(* POU GENERAL/xFctCheckNumber, ST *)
FUNCTION xFctCheckNumber : BOOL
VAR_INPUT
	sValue:STRING(255);
	xAlowDoubleSign:BOOL;
END_VAR
VAR
	iCharCount: INT;
	ii: INT;
	sCopyChar: STRING;
	xTmp: BOOL;
	xSyntaxError: BOOL;
	iCountPointChar: INT;
	iCountMinusChar: INT;
	iCountPlusChar: INT;
	iCountExponentChar: INT;
END_VAR
xFctCheckNumber:=FALSE;
iCharCount:=LEN(sValue);
iCountPointChar:=0;
iCountMinusChar:=0;
iCountPlusChar:=0;
iCountExponentChar:=0;
xSyntaxError:=FALSE;
IF (sValue <> '') THEN
	FOR ii:=1 TO iCharCount DO
		sCopyChar:=MID(sValue,1,ii);
		xTmp:=	(sCopyChar = '0') OR (sCopyChar = '1') OR (sCopyChar = '2') OR (sCopyChar = '3') OR (sCopyChar = '4') OR
				(sCopyChar = '5') OR (sCopyChar = '6') OR (sCopyChar = '7') OR (sCopyChar = '8') OR (sCopyChar = '9') OR
				(sCopyChar = '.') OR (sCopyChar = '-') OR (sCopyChar = '+') OR (sCopyChar = 'e') OR (sCopyChar = 'E');
		IF (sCopyChar = '.') THEN
			iCountPointChar:=iCountPointChar + 1;
		END_IF;
		IF (sCopyChar = '-') THEN
			iCountMinusChar:=iCountMinusChar + 1;
		END_IF;
		IF (sCopyChar = '+') THEN
			iCountPlusChar:=iCountPlusChar + 1;
		END_IF;
		IF (sCopyChar = 'e') OR (sCopyChar = 'E') THEN
			iCountExponentChar:=iCountExponentChar + 1;
			IF (iCountMinusChar > 0) THEN
				iCountMinusChar:=iCountMinusChar -1;
			END_IF;
			IF (iCountPlusChar > 0) THEN
				iCountPlusChar:=iCountPlusChar -1;
			END_IF;
		END_IF;
		IF NOT(xTmp) OR (iCountPointChar > 1) OR ((iCountMinusChar > 1) AND NOT(xAlowDoubleSign)) OR ((iCountMinusChar > 2) AND xAlowDoubleSign) OR
		    ((iCountPlusChar > 1) AND NOT(xAlowDoubleSign)) OR ((iCountPlusChar > 2) AND xAlowDoubleSign) OR (iCountExponentChar > 1) THEN
			xSyntaxError:=TRUE;
			EXIT;
		END_IF;
	END_FOR;
ELSE
	xSyntaxError:=TRUE;
END_IF;
xFctCheckNumber:=NOT(xSyntaxError);
END_FUNCTION

(* POU GENERAL/PROFILE/xFctCopyProfileToDataFile, ST *)
FUNCTION xFctCopyProfileToDataFile : BOOL
VAR_INPUT
	sNameOfProfile:STRING(30);
	ptrStProzessData:POINTER TO ST_EXCHG_PARAM_STANDARDPROCESS;
	ptrOnlineChangeData:POINTER TO ST_PROFILEONLINECHANGE_DATA;
	ptrDataFile:POINTER TO ARRAY[1..csiMaxFileLine] OF STRING(csiMaxCharPerLine);
END_VAR
VAR
(* variable *)
	i:INT;
(* Tmp *)
	sTmp:STRING;
END_VAR
(* Init. variable *)
	xFctCopyProfileToDataFile:=FALSE;
	i:=1;

(* copy value *)
	(* Name of the profile *)
		ptrDataFile^[i]:=sNameOfProfile;i:=i+1;
		sTmp:=CONCAT('001:rTorqueLevelHC:=',REAL_TO_STRING(ptrOnlineChangeData^.rTorqueLevelHC));
		ptrDataFile^[i]:=CONCAT(sTmp,';');i:=i+1;
		sTmp:=CONCAT('002:rForceDeflection:=',REAL_TO_STRING(ptrOnlineChangeData^.rForceDeflection));
		ptrDataFile^[i]:=CONCAT(sTmp,';');i:=i+1;
		sTmp:=CONCAT('003:rWorkingSpeedForward:=',REAL_TO_STRING(ptrOnlineChangeData^.rWorkingSpeedForward));
		ptrDataFile^[i]:=CONCAT(sTmp,';');i:=i+1;
		sTmp:=CONCAT('004:rWorkingOffsetBackward:=',REAL_TO_STRING(ptrOnlineChangeData^.rWorkingOffsetBackward));
		ptrDataFile^[i]:=CONCAT(sTmp,';');i:=i+1;
		sTmp:=CONCAT('005:rWorkingSpeedBackward:=',REAL_TO_STRING(ptrOnlineChangeData^.rWorkingSpeedBackward));
		ptrDataFile^[i]:=CONCAT(sTmp,';');i:=i+1;
		sTmp:=CONCAT('006:rWorkingSpindleSpeed:=',REAL_TO_STRING(ptrOnlineChangeData^.rWorkingSpindleSpeed));
		ptrDataFile^[i]:=CONCAT(sTmp,';');i:=i+1;

		sTmp:=CONCAT('007:rPositionLoad:=',REAL_TO_STRING(ptrStProzessData^.rPositionLoad));
		ptrDataFile^[i]:=CONCAT(sTmp,';');i:=i+1;
		sTmp:=CONCAT('008:rPositionStartProc:=',REAL_TO_STRING(ptrStProzessData^.rPositionStartProc));
		ptrDataFile^[i]:=CONCAT(sTmp,';');i:=i+1;
		sTmp:=CONCAT('009:rPositionEndProc:=',REAL_TO_STRING(ptrStProzessData^.rPositionEndProc));
		ptrDataFile^[i]:=CONCAT(sTmp,';');i:=i+1;
		sTmp:=CONCAT('010:rPositionToolChange:=',REAL_TO_STRING(ptrStProzessData^.rPositionToolChange));
		ptrDataFile^[i]:=CONCAT(sTmp,';');i:=i+1;
		sTmp:=CONCAT('011:rInfeedZAxisSpeed:=',REAL_TO_STRING(ptrStProzessData^.rInfeedZAxisSpeed));
		ptrDataFile^[i]:=CONCAT(sTmp,';');i:=i+1;
		sTmp:=CONCAT('012:rInfeedSpindleSpeed:=',REAL_TO_STRING(ptrStProzessData^.rInfeedSpindleSpeed));
		ptrDataFile^[i]:=CONCAT(sTmp,';');i:=i+1;
		sTmp:=CONCAT('013:rOutfeedStrokeAxisSpeed:=',REAL_TO_STRING(ptrStProzessData^.rOutfeedStrokeAxisSpeed));
		ptrDataFile^[i]:=CONCAT(sTmp,';');i:=i+1;
		sTmp:=CONCAT('014:rOutfeedSpindleSpeed:=',REAL_TO_STRING(ptrStProzessData^.rOutfeedSpindleSpeed));
		ptrDataFile^[i]:=CONCAT(sTmp,';');i:=i+1;
		sTmp:=CONCAT('015:rInfeedForceDeflection:=',REAL_TO_STRING(ptrStProzessData^.rInfeedForceDeflection));
		ptrDataFile^[i]:=CONCAT(sTmp,';');i:=i+1;
		sTmp:=CONCAT('016:rInfeedOffsetBackward:=',REAL_TO_STRING(ptrStProzessData^.rInfeedOffsetBackward));
		ptrDataFile^[i]:=CONCAT(sTmp,';');i:=i+1;
		sTmp:=CONCAT('017:iNumberTryInfeed:=',INT_TO_STRING(ptrStProzessData^.iNumberTryInfeed));
		ptrDataFile^[i]:=CONCAT(sTmp,';');i:=i+1;

		sTmp:=CONCAT('018:rProcessMinTime:=',REAL_TO_STRING(ptrStProzessData^.rProcessMinTime));
		ptrDataFile^[i]:=CONCAT(sTmp,';');i:=i+1;
		sTmp:=CONCAT('019:rProcessMaxTime:=',REAL_TO_STRING(ptrStProzessData^.rProcessMaxTime));
		ptrDataFile^[i]:=CONCAT(sTmp,';');i:=i+1;
		sTmp:=CONCAT('020:iHCStartProcPosCounter:=',INT_TO_STRING(ptrStProzessData^.iHCStartProcPosCounter));
		ptrDataFile^[i]:=CONCAT(sTmp,';');i:=i+1;
		sTmp:=CONCAT('021:rDeflectionSensorOffset:=',REAL_TO_STRING(ptrStProzessData^.rDeflectionSensorOffset));
		ptrDataFile^[i]:=CONCAT(sTmp,';');i:=i+1;
		sTmp:=CONCAT('022:rTorqueLevel_Overload:=',REAL_TO_STRING(ptrStProzessData^.rTorqueLevel_Overload));
		ptrDataFile^[i]:=CONCAT(sTmp,';');i:=i+1;

		sTmp:=CONCAT('023:iSparkOutStrokeCount:=',INT_TO_STRING(ptrStProzessData^.iSparkOutStrokeCount));
		ptrDataFile^[i]:=CONCAT(sTmp,';');i:=i+1;
		sTmp:=CONCAT('024:rSparkOutStrokeLength:=',REAL_TO_STRING(ptrStProzessData^.rSparkOutStrokeLength));
		ptrDataFile^[i]:=CONCAT(sTmp,';');i:=i+1;
		sTmp:=CONCAT('025:rSparkOutStrokeSpeed:=',REAL_TO_STRING(ptrStProzessData^.rSparkOutStrokeSpeed));
		ptrDataFile^[i]:=CONCAT(sTmp,';');i:=i+1;
		sTmp:=CONCAT('026:rSparkOutForceDeflection:=',REAL_TO_STRING(ptrStProzessData^.rSparkOutForceDeflection));
		ptrDataFile^[i]:=CONCAT(sTmp,';');i:=i+1;
		sTmp:=CONCAT('027:rSparkOutTorqueLevel:=',REAL_TO_STRING(ptrStProzessData^.rSparkOutTorqueLevel));
		ptrDataFile^[i]:=CONCAT(sTmp,';');i:=i+1;

		sTmp:=CONCAT('028:rPosToolGuid_Up:=',REAL_TO_STRING(ptrStProzessData^.rPosToolGuid_Up));
		ptrDataFile^[i]:=CONCAT(sTmp,';');i:=i+1;
		sTmp:=CONCAT('029:rPosToolGuid_Down:=',REAL_TO_STRING(ptrStProzessData^.rPosToolGuid_Down));
		ptrDataFile^[i]:=CONCAT(sTmp,';');i:=i+1;
		sTmp:=CONCAT('030:rDistanceToolGuide:=',REAL_TO_STRING(ptrStProzessData^.rDistanceToolGuide));
		ptrDataFile^[i]:=CONCAT(sTmp,';');i:=i+1;
		sTmp:=CONCAT('031:rDistanceToolEndPos:=',REAL_TO_STRING(ptrStProzessData^.rDistanceToolEndPos));
		ptrDataFile^[i]:=CONCAT(sTmp,';');i:=i+1;
		sTmp:=CONCAT('032:rLengthTool_Fixed:=',REAL_TO_STRING(ptrStProzessData^.rLengthTool_Fixed));
		ptrDataFile^[i]:=CONCAT(sTmp,';');i:=i+1;
		sTmp:=CONCAT('033:rLengthTool_Work:=',REAL_TO_STRING(ptrStProzessData^.rLengthTool_Work));
		ptrDataFile^[i]:=CONCAT(sTmp,';');i:=i+1;
		sTmp:=CONCAT('034:rLengthToolGuide:=',REAL_TO_STRING(ptrStProzessData^.rLengthToolGuide));
		ptrDataFile^[i]:=CONCAT(sTmp,';');i:=i+1;
		sTmp:=CONCAT('035:rLengthAirTableBoard:=',REAL_TO_STRING(ptrStProzessData^.rLengthAirTableBoard));
		ptrDataFile^[i]:=CONCAT(sTmp,';');i:=i+1;
		sTmp:=CONCAT('036:xConfigActive:=',BOOL_TO_STRING(ptrStProzessData^.xConfigActive));
		ptrDataFile^[i]:=CONCAT(sTmp,';');i:=i+1;

		sTmp:=CONCAT('037:iMaxTorque:=',INT_TO_STRING(ptrStProzessData^.iMaxTorque));
		ptrDataFile^[i]:=CONCAT(sTmp,';');i:=i+1;
		sTmp:=CONCAT('038:rSpeedZAxisForBackward:=',REAL_TO_STRING(ptrStProzessData^.rSpeedZAxisForBackward));
		ptrDataFile^[i]:=CONCAT(sTmp,';');i:=i+1;
		sTmp:=CONCAT('039:rWorkingSpeedOscillation:=',REAL_TO_STRING(ptrStProzessData^.rWorkingSpeedOscillation));
		ptrDataFile^[i]:=CONCAT(sTmp,';');i:=i+1;
		sTmp:=CONCAT('040:rZ1AxisPosSwitchOAxisOff:=',REAL_TO_STRING(ptrStProzessData^.rZ1AxisPosSwitchOAxisOff));
		ptrDataFile^[i]:=CONCAT(sTmp,';');i:=i+1;
		sTmp:=CONCAT('041:xActivateCoolantProcess:=',BOOL_TO_STRING(ptrStProzessData^.xActivateCoolantProcess));
		ptrDataFile^[i]:=CONCAT(sTmp,';');i:=i+1;
		sTmp:=CONCAT('042:rStrokeAxisPosSwitchCoolantOff:=',REAL_TO_STRING(ptrStProzessData^.rStrokeAxisPosSwitchCoolantOff));
		ptrDataFile^[i]:=CONCAT(sTmp,';');i:=i+1;

		sTmp:=CONCAT('043:rCentringPosZ1Axis:=',REAL_TO_STRING(ptrStProzessData^.rCentringPosZ1Axis));
		ptrDataFile^[i]:=CONCAT(sTmp,';');i:=i+1;
		sTmp:=CONCAT('044:rCentringPosSpeedSlowZ1Axis:=',REAL_TO_STRING(ptrStProzessData^.rCentringPosSpeedSlowZ1Axis));
		ptrDataFile^[i]:=CONCAT(sTmp,';');i:=i+1;
		sTmp:=CONCAT('045:rCentringPosSpeedFastZ1Axis:=',REAL_TO_STRING(ptrStProzessData^.rCentringPosSpeedFastZ1Axis));
		ptrDataFile^[i]:=CONCAT(sTmp,';');i:=i+1;
		sTmp:=CONCAT('046:rCentringSpeedSAxis:=',REAL_TO_STRING(ptrStProzessData^.rCentringSpeedSAxis));
		ptrDataFile^[i]:=CONCAT(sTmp,';');i:=i+1;
		sTmp:=CONCAT('047:rCentringSpeedOAxis:=',REAL_TO_STRING(ptrStProzessData^.rCentringSpeedOAxis));
		ptrDataFile^[i]:=CONCAT(sTmp,';');i:=i+1;
		sTmp:=CONCAT('048:rCentringBackStrokeOffsetFirstHC:=',REAL_TO_STRING(ptrStProzessData^.rCentringBackStrokeOffsetFirstHC));
		ptrDataFile^[i]:=CONCAT(sTmp,';');i:=i+1;
		sTmp:=CONCAT('049:rCentringBackStrokeOffsetAfterFirstHC:=',REAL_TO_STRING(ptrStProzessData^.rCentringBackStrokeOffsetAfterFirstHC));
		ptrDataFile^[i]:=CONCAT(sTmp,';');i:=i+1;
		sTmp:=CONCAT('050:rCentringOffsetBeforeLastHC:=',REAL_TO_STRING(ptrStProzessData^.rCentringOffsetBeforeLastHC));
		ptrDataFile^[i]:=CONCAT(sTmp,';');i:=i+1;
		sTmp:=CONCAT('051:rCentringBackStrokeSpeed:=',REAL_TO_STRING(ptrStProzessData^.rCentringBackStrokeSpeed));
		ptrDataFile^[i]:=CONCAT(sTmp,';');i:=i+1;
		sTmp:=CONCAT('052:rCentringTimeHCActive:=',REAL_TO_STRING(ptrStProzessData^.rCentringTimeHCActive));
		ptrDataFile^[i]:=CONCAT(sTmp,';');i:=i+1;
		sTmp:=CONCAT('053:rCentringTimeHCInactive:=',REAL_TO_STRING(ptrStProzessData^.rCentringTimeHCInactive));
		ptrDataFile^[i]:=CONCAT(sTmp,';');i:=i+1;
		sTmp:=CONCAT('054:iCentringNumberMaxHCinWindow:=',INT_TO_STRING(ptrStProzessData^.iCentringNumberMaxHCinWindow));
		ptrDataFile^[i]:=CONCAT(sTmp,';');i:=i+1;
		sTmp:=CONCAT('055:rCentringHCWindow:=',REAL_TO_STRING(ptrStProzessData^.rCentringHCWindow));
		ptrDataFile^[i]:=CONCAT(sTmp,';');i:=i+1;
		sTmp:=CONCAT('056:rCentringForceDeflection:=',REAL_TO_STRING(ptrStProzessData^.rCentringForceDeflection));
		ptrDataFile^[i]:=CONCAT(sTmp,';');i:=i+1;
		sTmp:=CONCAT('057:rCentringOffsetBackward:=',REAL_TO_STRING(ptrStProzessData^.rCentringOffsetBackward));
		ptrDataFile^[i]:=CONCAT(sTmp,';');i:=i+1;
		sTmp:=CONCAT('058:rCenteringDeflectionSensorOffset:=',REAL_TO_STRING(ptrStProzessData^.rCenteringDeflectionSensorOffset));
		ptrDataFile^[i]:=CONCAT(sTmp,';');i:=i+1;
		sTmp:=CONCAT('059:rCentringOffsetSlowToFastZSpeed:=',REAL_TO_STRING(ptrStProzessData^.rCentringOffsetSlowToFastZSpeed));
		ptrDataFile^[i]:=CONCAT(sTmp,';');i:=i+1;
		sTmp:=CONCAT('060:iCentringSelectProcess:=',INT_TO_STRING(ptrStProzessData^.iCentringSelectProcess));
		ptrDataFile^[i]:=CONCAT(sTmp,';');i:=i+1;
		sTmp:=CONCAT('061:xPositionEndProcIncOnOff:=',BOOL_TO_STRING(ptrStProzessData^.xPositionEndProcIncOnOff));
		ptrDataFile^[i]:=CONCAT(sTmp,';');i:=i+1;
		sTmp:=CONCAT('062:rPositionEndProcMaxInc:=',REAL_TO_STRING(ptrStProzessData^.rPositionEndProcMaxInc));
		ptrDataFile^[i]:=CONCAT(sTmp,';');i:=i+1;
		sTmp:=CONCAT('063:rPositionEndProInc:=',REAL_TO_STRING(ptrStProzessData^.rPositionEndProInc));
		ptrDataFile^[i]:=CONCAT(sTmp,';');i:=i+1;

		sTmp:=CONCAT('064:iWorkControlType:=',INT_TO_STRING(ptrStProzessData^.iWorkControlType));
		ptrDataFile^[i]:=CONCAT(sTmp,';');i:=i+1;
		sTmp:=CONCAT('065:rZ_PID_Torque:=',REAL_TO_STRING(ptrStProzessData^.rZ_PID_Torque));
		ptrDataFile^[i]:=CONCAT(sTmp,';');i:=i+1;
		sTmp:=CONCAT('066:rZ_PID_MinSpeed:=',REAL_TO_STRING(ptrStProzessData^.rZ_PID_MinSpeed));
		ptrDataFile^[i]:=CONCAT(sTmp,';');i:=i+1;
		sTmp:=CONCAT('067:rZ_PID_MaxSpeed:=',REAL_TO_STRING(ptrStProzessData^.rZ_PID_MaxSpeed));
		ptrDataFile^[i]:=CONCAT(sTmp,';');i:=i+1;
		sTmp:=CONCAT('068:rZ_PID_Kp:=',REAL_TO_STRING(ptrStProzessData^.rZ_PID_Kp));
		ptrDataFile^[i]:=CONCAT(sTmp,';');i:=i+1;
		sTmp:=CONCAT('069:rZ_PID_Ki:=',REAL_TO_STRING(ptrStProzessData^.rZ_PID_Ki));
		ptrDataFile^[i]:=CONCAT(sTmp,';');i:=i+1;
		sTmp:=CONCAT('070:rZ_PID_Kd:=',REAL_TO_STRING(ptrStProzessData^.rZ_PID_Kd));
		ptrDataFile^[i]:=CONCAT(sTmp,';');i:=i+1;
		sTmp:=CONCAT('071:iZ_PID_FilterM:=',INT_TO_STRING(ptrStProzessData^.iZ_PID_FilterM));
		ptrDataFile^[i]:=CONCAT(sTmp,';');i:=i+1;
		sTmp:=CONCAT('072:rZ_D_Kd:=',REAL_TO_STRING(ptrStProzessData^.rZ_D_Kd));
		ptrDataFile^[i]:=CONCAT(sTmp,';');i:=i+1;
		sTmp:=CONCAT('073:iZ_D_FilterM:=',INT_TO_STRING(ptrStProzessData^.iZ_D_FilterM));
		ptrDataFile^[i]:=CONCAT(sTmp,';');i:=i+1;

		sTmp:=CONCAT('074:rSuspensionBubblerSpeed:=',REAL_TO_STRING(ptrStProzessData^.rSuspensionBubblerSpeed));
		ptrDataFile^[i]:=CONCAT(sTmp,';');i:=i+1;
		sTmp:=CONCAT('075:rSuspensionFeederSpeed:=',REAL_TO_STRING(ptrStProzessData^.rSuspensionFeederSpeed));
		ptrDataFile^[i]:=CONCAT(sTmp,';');i:=i+1;

		sTmp:=CONCAT('076:rOutfeedStrokeAxisSpeedSlow:=',REAL_TO_STRING(ptrStProzessData^.rOutfeedStrokeAxisSpeedSlow));
		ptrDataFile^[i]:=CONCAT(sTmp,';');i:=i+1;
		sTmp:=CONCAT('077:rZ1AxisPosSwitchFastVel:=',REAL_TO_STRING(ptrStProzessData^.rZ1AxisPosSwitchFastVel));
		ptrDataFile^[i]:=CONCAT(sTmp,';');i:=i+1;
		sTmp:=CONCAT('078:rZ1AxisOffsetStartRecordTorque:=',REAL_TO_STRING(ptrStProzessData^.rZ1AxisOffsetStartRecordTorque));
		ptrDataFile^[i]:=CONCAT(sTmp,';');i:=i+1;

		sTmp:=CONCAT('079:xCentringEndProcIncOnOff:=',BOOL_TO_STRING(ptrStProzessData^.xCentringEndProcIncOnOff));
		ptrDataFile^[i]:=CONCAT(sTmp,';');i:=i+1;
		sTmp:=CONCAT('080:rCentringEndProInc:=',REAL_TO_STRING(ptrStProzessData^.rCentringEndProInc));
		ptrDataFile^[i]:=CONCAT(sTmp,';');i:=i+1;

		sTmp:=CONCAT('081:rWorkingSpindleSpeedMinMax:=',REAL_TO_STRING(ptrStProzessData^.rWorkingSpindleSpeedMinMax));
		ptrDataFile^[i]:=CONCAT(sTmp,';');i:=i+1;
		sTmp:=CONCAT('082:rO_Ctrl_TorquePercent_OFF:=',REAL_TO_STRING(ptrStProzessData^.rO_Ctrl_TorquePercent_OFF));
		ptrDataFile^[i]:=CONCAT(sTmp,';');i:=i+1;
		sTmp:=CONCAT('083:rO_Ctrl_HystereseOffset:=',REAL_TO_STRING(ptrStProzessData^.rO_Ctrl_HystereseOffset));
		ptrDataFile^[i]:=CONCAT(sTmp,';');i:=i+1;

		sTmp:=CONCAT('084:rZPositionCylindricalArea:=',REAL_TO_STRING(ptrStProzessData^.rZPositionCylindricalArea));
		ptrDataFile^[i]:=CONCAT(sTmp,';');i:=i+1;
		sTmp:=CONCAT('085:rZMinThresholdTroqueEndProcess:=',REAL_TO_STRING(ptrStProzessData^.rZMinThresholdTroqueEndProcess));
		ptrDataFile^[i]:=CONCAT(sTmp,';');i:=i+1;

		sTmp:=CONCAT('086:rDistProgressStroke:=',REAL_TO_STRING(ptrStProzessData^.rDistProgressStroke));
		ptrDataFile^[i]:=CONCAT(sTmp,';');i:=i+1;
		sTmp:=CONCAT('087:iProgressStrokeStartTorque:=',INT_TO_STRING(ptrStProzessData^.iProgressStrokeStartTorque));
		ptrDataFile^[i]:=CONCAT(sTmp,';');i:=i+1;
		sTmp:=CONCAT('088:rProgressStrokeStopOffset:=',REAL_TO_STRING(ptrStProzessData^.rProgressStrokeStopOffset));
		ptrDataFile^[i]:=CONCAT(sTmp,';');i:=i+1;
		sTmp:=CONCAT('089:iCleanNozzleMode:=',INT_TO_STRING(ptrStProzessData^.iCleanNozzleMode));
		ptrDataFile^[i]:=CONCAT(sTmp,';');i:=i+1;
		sTmp:=CONCAT('090:ioutfeedstrokecontroller:=',INT_TO_STRING(ptrStProzessData^.iOutfeedStrokeController));
		ptrDataFile^[i]:=CONCAT(sTmp,';');i:=i+1;
		sTmp:=CONCAT('091:isparkoutcontroller:=',INT_TO_STRING(ptrStProzessData^.iSparkOutController));
		ptrDataFile^[i]:=CONCAT(sTmp,';');i:=i+1;

	(* add empty line to set the end *)
	ptrDataFile^[i]:='';

	(* confirm copy *)
	xFctCopyProfileToDataFile:=TRUE;
END_FUNCTION

(* POU GENERAL/PROFILE/xFctSetDefaultValueStaticProfile, ST *)
FUNCTION xFctSetDefaultValueStaticProfile : BOOL
VAR_INPUT
	ptrT_DefaultProfileParameter:POINTER TO ARRAY [1..1] OF ST_RETAIN_DATA_PROFILEPARAMETER;
END_VAR
VAR
(* variable *)
	ii:INT;
END_VAR
	(* Init. value *)
	xFctSetDefaultValueStaticProfile:=FALSE;
	FOR ii:=1 TO 1 DO
		ptrT_DefaultProfileParameter^[ii].T_ProfileOnlineChange.rTorqueLevelHC:=80.0;
		ptrT_DefaultProfileParameter^[ii].T_ProfileOnlineChange.rForceDeflection:=18.0;
		ptrT_DefaultProfileParameter^[ii].T_ProfileOnlineChange.rWorkingSpeedForward:=100.0;
		ptrT_DefaultProfileParameter^[ii].T_ProfileOnlineChange.rWorkingOffsetBackward:=0.0;
		ptrT_DefaultProfileParameter^[ii].T_ProfileOnlineChange.rWorkingSpeedBackward:=0.5;
		ptrT_DefaultProfileParameter^[ii].T_ProfileOnlineChange.rWorkingSpindleSpeed:=6000.0;

		ptrT_DefaultProfileParameter^[ii].T_ProzessData.rPositionLoad:=-446.0;
		ptrT_DefaultProfileParameter^[ii].T_ProzessData.rPositionStartProc:=-410.0;
		ptrT_DefaultProfileParameter^[ii].T_ProzessData.rPositionEndProc:=-80.0;
		ptrT_DefaultProfileParameter^[ii].T_ProzessData.rPositionToolChange:=-510.0;
		ptrT_DefaultProfileParameter^[ii].T_ProzessData.rInfeedZAxisSpeed:=50.0;
		ptrT_DefaultProfileParameter^[ii].T_ProzessData.rInfeedSpindleSpeed:=500.0;
		ptrT_DefaultProfileParameter^[ii].T_ProzessData.rOutfeedStrokeAxisSpeed:=250.0;
		ptrT_DefaultProfileParameter^[ii].T_ProzessData.rOutfeedSpindleSpeed:=500.0;
		ptrT_DefaultProfileParameter^[ii].T_ProzessData.rInfeedForceDeflection:=5.0;
		ptrT_DefaultProfileParameter^[ii].T_ProzessData.rInfeedOffsetBackward:=-10.0;
		ptrT_DefaultProfileParameter^[ii].T_ProzessData.iNumberTryInfeed:=5;

		ptrT_DefaultProfileParameter^[ii].T_ProzessData.rProcessMinTime:=5.0;
		ptrT_DefaultProfileParameter^[ii].T_ProzessData.rProcessMaxTime:=120.0;
		ptrT_DefaultProfileParameter^[ii].T_ProzessData.iHCStartProcPosCounter:=3;
		ptrT_DefaultProfileParameter^[ii].T_ProzessData.rDeflectionSensorOffset:=0.2;
		ptrT_DefaultProfileParameter^[ii].T_ProzessData.rTorqueLevel_Overload:=60.0;

		ptrT_DefaultProfileParameter^[ii].T_ProzessData.iSparkOutStrokeCount:=2;
		ptrT_DefaultProfileParameter^[ii].T_ProzessData.rSparkOutStrokeLength:=-20.0;
		ptrT_DefaultProfileParameter^[ii].T_ProzessData.rSparkOutStrokeSpeed:=200.0;
		ptrT_DefaultProfileParameter^[ii].T_ProzessData.rSparkOutForceDeflection:=80.0;
		ptrT_DefaultProfileParameter^[ii].T_ProzessData.rSparkOutTorqueLevel:=20.0;

		ptrT_DefaultProfileParameter^[ii].T_ProzessData.rPosToolGuid_Up:=210;
		ptrT_DefaultProfileParameter^[ii].T_ProzessData.rPosToolGuid_Down:=185;
		ptrT_DefaultProfileParameter^[ii].T_ProzessData.rDistanceToolGuide:=4.5;
		ptrT_DefaultProfileParameter^[ii].T_ProzessData.rDistanceToolEndPos:=4.5;
		ptrT_DefaultProfileParameter^[ii].T_ProzessData.rLengthTool_Fixed:=450.0;
		ptrT_DefaultProfileParameter^[ii].T_ProzessData.rLengthTool_Work:=325.0;
		ptrT_DefaultProfileParameter^[ii].T_ProzessData.rLengthToolGuide:=10.0;
		ptrT_DefaultProfileParameter^[ii].T_ProzessData.rLengthAirTableBoard:=33.0;
		ptrT_DefaultProfileParameter^[ii].T_ProzessData.xConfigActive:=FALSE;

		ptrT_DefaultProfileParameter^[ii].T_ProzessData.iMaxTorque:=130;
		ptrT_DefaultProfileParameter^[ii].T_ProzessData.rSpeedZAxisForBackward:=1.0;
		ptrT_DefaultProfileParameter^[ii].T_ProzessData.rWorkingSpeedOscillation:=0.0;
		ptrT_DefaultProfileParameter^[ii].T_ProzessData.rZ1AxisPosSwitchOAxisOff:=0.0;
		ptrT_DefaultProfileParameter^[ii].T_ProzessData.xActivateCoolantProcess:=FALSE;
		ptrT_DefaultProfileParameter^[ii].T_ProzessData.rStrokeAxisPosSwitchCoolantOff:=-300.0;

		ptrT_DefaultProfileParameter^[ii].T_ProzessData.rCentringPosZ1Axis:=-400.0;
		ptrT_DefaultProfileParameter^[ii].T_ProzessData.rCentringPosSpeedSlowZ1Axis:=20.0;
		ptrT_DefaultProfileParameter^[ii].T_ProzessData.rCentringPosSpeedFastZ1Axis:=50.0;
		ptrT_DefaultProfileParameter^[ii].T_ProzessData.rCentringSpeedSAxis:=500.0;
		ptrT_DefaultProfileParameter^[ii].T_ProzessData.rCentringSpeedOAxis:=40.0;
		ptrT_DefaultProfileParameter^[ii].T_ProzessData.rCentringBackStrokeOffsetFirstHC:=-5.0;
		ptrT_DefaultProfileParameter^[ii].T_ProzessData.rCentringBackStrokeOffsetAfterFirstHC:=-15.0;
		ptrT_DefaultProfileParameter^[ii].T_ProzessData.rCentringOffsetBeforeLastHC:=-3.0;
		ptrT_DefaultProfileParameter^[ii].T_ProzessData.rCentringBackStrokeSpeed:=10.0;
		ptrT_DefaultProfileParameter^[ii].T_ProzessData.rCentringTimeHCActive:=5.0;
		ptrT_DefaultProfileParameter^[ii].T_ProzessData.rCentringTimeHCInactive:=0.5;
		ptrT_DefaultProfileParameter^[ii].T_ProzessData.iCentringNumberMaxHCinWindow:=5;
		ptrT_DefaultProfileParameter^[ii].T_ProzessData.rCentringHCWindow:=0.5;
		ptrT_DefaultProfileParameter^[ii].T_ProzessData.rCentringForceDeflection:=20.0;
		ptrT_DefaultProfileParameter^[ii].T_ProzessData.rCentringOffsetBackward:=-1.0;
		ptrT_DefaultProfileParameter^[ii].T_ProzessData.rCenteringDeflectionSensorOffset:=0.3;
		ptrT_DefaultProfileParameter^[ii].T_ProzessData.rCentringOffsetSlowToFastZSpeed:=40.0;
		ptrT_DefaultProfileParameter^[ii].T_ProzessData.iCentringSelectProcess:=1;
		ptrT_DefaultProfileParameter^[ii].T_ProzessData.xPositionEndProcIncOnOff:=0;
		ptrT_DefaultProfileParameter^[ii].T_ProzessData.rPositionEndProcMaxInc:=-10.0;
		ptrT_DefaultProfileParameter^[ii].T_ProzessData.rPositionEndProInc:=0.2;
		ptrT_DefaultProfileParameter^[ii].T_ProzessData.rOutfeedStrokeAxisSpeedSlow:=2.0;
		ptrT_DefaultProfileParameter^[ii].T_ProzessData.rZ1AxisPosSwitchFastVel:=0.0;
		ptrT_DefaultProfileParameter^[ii].T_ProzessData.rZ1AxisOffsetStartRecordTorque:=0.0;
		ptrT_DefaultProfileParameter^[ii].T_ProzessData.xCentringEndProcIncOnOff:=0;
		ptrT_DefaultProfileParameter^[ii].T_ProzessData.rCentringEndProInc:=0.2;
		ptrT_DefaultProfileParameter^[ii].T_ProzessData.rWorkingSpindleSpeedMinMax:=6000.0;
		ptrT_DefaultProfileParameter^[ii].T_ProzessData.rO_Ctrl_TorquePercent_OFF:=100.0;
		ptrT_DefaultProfileParameter^[ii].T_ProzessData.rO_Ctrl_HystereseOffset:=10.0;
		ptrT_DefaultProfileParameter^[ii].T_ProzessData.rZPositionCylindricalArea:=-240.0;
		ptrT_DefaultProfileParameter^[ii].T_ProzessData.rZMinThresholdTroqueEndProcess:=12.0;

		ptrT_DefaultProfileParameter^[ii].T_ProzessData.iWorkControlType:=1;
		ptrT_DefaultProfileParameter^[ii].T_ProzessData.rZ_PID_Torque:=50.0;
		ptrT_DefaultProfileParameter^[ii].T_ProzessData.rZ_PID_MinSpeed:=2.0;
		ptrT_DefaultProfileParameter^[ii].T_ProzessData.rZ_PID_MaxSpeed:=40.0;
		ptrT_DefaultProfileParameter^[ii].T_ProzessData.rZ_PID_Kp:=2.0;
		ptrT_DefaultProfileParameter^[ii].T_ProzessData.rZ_PID_Ki:=0.5;
		ptrT_DefaultProfileParameter^[ii].T_ProzessData.rZ_PID_Kd:=0.01;
		ptrT_DefaultProfileParameter^[ii].T_ProzessData.iZ_PID_FilterM:=20;
		ptrT_DefaultProfileParameter^[ii].T_ProzessData.rZ_D_Kd:=0.01;
		ptrT_DefaultProfileParameter^[ii].T_ProzessData.iZ_D_FilterM:=20;

		ptrT_DefaultProfileParameter^[ii].T_ProzessData.rSuspensionBubblerSpeed:=20.0;
		ptrT_DefaultProfileParameter^[ii].T_ProzessData.rSuspensionFeederSpeed:=20.0;

		ptrT_DefaultProfileParameter^[ii].T_ProzessData.rDistProgressStroke:=0.0;
		ptrT_DefaultProfileParameter^[ii].T_ProzessData.iProgressStrokeStartTorque:=0;
		ptrT_DefaultProfileParameter^[ii].T_ProzessData.rProgressStrokeStopOffset:=0.0;
		ptrT_DefaultProfileParameter^[ii].T_ProzessData.iCleanNozzleMode:=0;
		ptrT_DefaultProfileParameter^[ii].T_ProzessData.iOutfeedStrokeController:=0;
		ptrT_DefaultProfileParameter^[ii].T_ProzessData.iSparkOutController:=0;

	END_FOR;
	(* Confirm Default setting *)
	xFctSetDefaultValueStaticProfile:=TRUE;
END_FUNCTION

(* POU GENERAL/FB_PASSWORD, ST *)
FUNCTION_BLOCK FB_PASSWORD
VAR_INPUT
END_VAR
VAR_IN_OUT
	T_Password:ST_PASSWORD;
	T_HDD:ST_HDD;
END_VAR
VAR_OUTPUT
END_VAR
VAR
	RisingEdgeReset: R_TRIG;
	xConfirmResetFB: BOOL;
	TimerFileLocked: TON;
	RisingEdgeExecute: R_TRIG;
	TimerOut: TON;
	xTmp: BOOL;
	tTimeOut: TIME;
	iStepFunction: INT;
	xReadPassword: BOOL;
	sDeleteData: ARRAY[1..csiMaxFileLine] OF STRING(csiMaxCharPerLine);
	sTmp:STRING(255);
	xWritePassword: BOOL;
END_VAR
(****************************************************************************************************************************************************)
(***********                            	      This Functionblock read and write the Operator Password from a File                		    ************)
(****************************************************************************************************************************************************)
(* waiting for reset *)
	RisingEdgeReset(CLK:=T_Password.T_Ctrle.xReset);
	IF RisingEdgeReset.Q THEN
	(* init. structure *)
		T_Password.T_Ctrle.xDone:=FALSE;
		T_Password.T_Ctrle.xErr:=FALSE;
		T_Password.T_Ctrle.udiErrorID:=0;
		T_Password.T_Ctrle.iFunction:=0;
		(* Reset HDD if error activ *)
		IF T_HDD.T_Ctrle.xErr THEN T_HDD.T_Ctrle.xReset:=TRUE; END_IF
		(* Init. variable *)
		xReadPassword:=FALSE;
		xWritePassword:=FALSE;
		(* set flag done *)
		xConfirmResetFB:=TRUE;
		(* exit function *)
		RETURN;
	ELSE
		IF xConfirmResetFB THEN
		(* confirm reset FB *)
			T_Password.T_Ctrle.xDone:=TRUE;
			T_Password.T_Ctrle.xErr:=FALSE;
			T_Password.T_Ctrle.udiErrorID:=0;
			T_Password.T_Ctrle.iFunction:=0;
			(* init. variable *)
			xConfirmResetFB:=FALSE;
		END_IF
	END_IF

TimerFileLocked(IN:=TRUE, PT:=T#10S);

(* waiting for execute *)
	RisingEdgeExecute(CLK:=T_Password.T_Ctrle.xExecute);
	IF RisingEdgeExecute.Q THEN
		CASE T_Password.T_Ctrle.iFunction OF
		(* read Operator Password *)
		1:	xReadPassword:=TRUE;
			T_HDD.T_Data.sData:=sDeleteData;
			tTimeOut:=T#10s;
		(* write Operator Password *)
		2:	xWritePassword:=TRUE;
			T_HDD.T_Data.sData:=sDeleteData;
			tTimeOut:=T#10s;
		ELSE
		(* function not implemented *)
			 T_Password.T_Ctrle.xDone:=FALSE;
			 T_Password.T_Ctrle.xErr:=TRUE;
			 T_Password.T_Ctrle.udiErrorID:=16#F000;
			 (* exit FB *)
			 RETURN;
		END_CASE
		(* Init. variable *)
		T_Password.T_Ctrle.xDone:=FALSE;
		T_Password.T_Ctrle.xErr:=FALSE;
		T_Password.T_Ctrle.udiErrorID:=16#0;
		(* init. step *)
		iStepFunction:=1;
		RETURN;
	END_IF

(* Monitor time out *)
	xTmp:=	NOT T_Password.T_Ctrle.xDone
			AND NOT T_Password.T_Ctrle.xErr;
	TimerOut(IN:=xTmp, PT:=tTimeOut);
	IF TimerOut.Q THEN iStepFunction:=99; END_IF

(* read Operator Password *)
	IF xReadPassword THEN
		CASE iStepFunction OF
		(* start timeout *)
		1:	TimerFileLocked(IN:=FALSE);
			T_Password.T_Ctrle.udiGetOperatorPassword:=123456;
			T_Password.T_Ctrle.sGetOperatorPassword:='123456';
			iStepFunction:=iStepFunction + 1;
		(* file name and activ read or write *)
		2:	IF T_HDD.T_Ctrle.xDone AND NOT(T_HDD.T_Ctrle.xErr) AND NOT(T_HDD.T_Ctrle.xLocked) THEN
				sTmp:=CONCAT(cssRootPLC,'Bore800\Password\OperatorPassword.txt');
			(* activ read *)
				T_HDD.T_Ctrle.iFunction:=1;
				T_HDD.T_Ctrle.xLocked:=TRUE;
				T_HDD.T_File.sPathAndFileName:=sTmp;
				T_HDD.T_Ctrle.xExecute:=TRUE;
				(* next step *)
				iStepFunction:=iStepFunction + 1;
			ELSE
				(* activ error if time out done, HDD not ready *)
				IF TimerFileLocked.Q THEN
					 iStepFunction:=90;
				END_IF
			END_IF;
		(* waiting flag *)
		3:	IF T_HDD.T_Ctrle.xDone AND NOT(T_HDD.T_Ctrle.xErr) THEN iStepFunction:=iStepFunction + 1; END_IF
			IF T_HDD.T_Ctrle.xErr THEN T_HDD.T_Ctrle.xReset:=TRUE; iStepFunction:=5; END_IF
		(* check syntax *)
		4:	IF (FIND(STR1:=T_HDD.T_Data.sData[1],STR2:=';') > 0) THEN
				sTmp:=T_HDD.T_Data.sData[1];
				sTmp:=sFctDeleteChar(sString:=sTmp, sChar:='$N');
				sTmp:=sFctDeleteChar(sString:=sTmp, sChar:='$L');
				sTmp:=sFctDeleteChar(sString:=sTmp, sChar:=';');
				IF xFctCheckNumber(sValue:=sTmp,xAlowDoubleSign:=FALSE) THEN
				(* Syntax correct *)
					T_Password.T_Ctrle.sGetOperatorPassword:=sTmp;
					T_Password.T_Ctrle.udiGetOperatorPassword:=STRING_TO_UDINT(T_Password.T_Ctrle.sGetOperatorPassword);
					iStepFunction:=90;
				ELSE
					(* Wrong Syntax *)
					iStepFunction:=10;	(* Create new File *)
				END_IF;
			ELSE
				(* Wrong Syntax *)
				iStepFunction:=10;	(* Create new File *)
			END_IF;
		5:	IF NOT(T_HDD.T_Ctrle.xReset) AND T_HDD.T_Ctrle.xDone THEN
				iStepFunction:=iStepFunction + 1;
			END_IF
		(* Create FirstLevel directory *)
		6:	sTmp:=CONCAT(cssRootPLC,'Bore800\');
			(* activ read *)
			T_HDD.T_Ctrle.iFunction:=7;
			T_HDD.T_File.sDirectoryPath:=sTmp;
			T_HDD.T_Ctrle.xExecute:=TRUE;
			(* next step *)
			iStepFunction:=iStepFunction + 1;
		(* waiting flag *)
		7:	IF T_HDD.T_Ctrle.xDone AND NOT(T_HDD.T_Ctrle.xErr) THEN iStepFunction:=iStepFunction + 1; END_IF
			IF T_HDD.T_Ctrle.xErr THEN T_HDD.T_Ctrle.xReset:=TRUE; iStepFunction:=iStepFunction + 1; END_IF
		(* Create SecondLevel directory *)
		8:	IF NOT(T_HDD.T_Ctrle.xReset) AND T_HDD.T_Ctrle.xDone THEN
				sTmp:=CONCAT(cssRootPLC,'Bore800\Password\');
				(* activ read *)
				T_HDD.T_Ctrle.iFunction:=7;
				T_HDD.T_File.sDirectoryPath:=sTmp;
				T_HDD.T_Ctrle.xExecute:=TRUE;
				(* next step *)
				iStepFunction:=iStepFunction + 1;
			END_IF;
		(* waiting flag *)
		9:	IF T_HDD.T_Ctrle.xDone AND NOT(T_HDD.T_Ctrle.xErr) THEN iStepFunction:=iStepFunction + 1; END_IF
			IF T_HDD.T_Ctrle.xErr THEN T_HDD.T_Ctrle.xReset:=TRUE; iStepFunction:=iStepFunction + 1; END_IF
		(* Create Password File *)
		10:	IF NOT(T_HDD.T_Ctrle.xReset) AND T_HDD.T_Ctrle.xDone THEN
				T_HDD.T_Data.sData:=sDeleteData;
				T_HDD.T_Data.sData[1]:='123456;';	(* Set Default Password *)
				T_Password.T_Ctrle.udiGetOperatorPassword:=123456;
				T_Password.T_Ctrle.sGetOperatorPassword:='123456';
				sTmp:=CONCAT(cssRootPLC,'Bore800\Password\OperatorPassword.txt');
				T_HDD.T_File.sPathAndFileName:=sTmp;
				T_HDD.T_Ctrle.iFunction:=2;
				T_HDD.T_Ctrle.xExecute:=TRUE;
				(* next step *)
				iStepFunction:=iStepFunction + 1;
			END_IF;
		(* waiting flag *)
		11:	IF T_HDD.T_Ctrle.xDone AND NOT(T_HDD.T_Ctrle.xErr) THEN iStepFunction:=90; END_IF
			IF T_HDD.T_Ctrle.xErr THEN iStepFunction:=80; END_IF
		(* reset error *)
		80:	T_HDD.T_Ctrle.xReset:=TRUE;
			iStepFunction:=91;
		(* done *)
		90:	T_Password.T_Ctrle.xDone:=TRUE;
			T_Password.T_Ctrle.xErr:=FALSE;
			T_Password.T_Ctrle.udiErrorID:=16#0;
			T_HDD.T_Ctrle.xLocked:=FALSE;
			xReadPassword:=FALSE;
		(* start read error *)
		91:	T_Password.T_Ctrle.xDone:=FALSE;
			T_Password.T_Ctrle.xErr:=TRUE;
			T_Password.T_Ctrle.udiErrorID:=16#F1000 + T_Password.T_Ctrle.iFunction;
			T_HDD.T_Ctrle.xReset:=T_HDD.T_Ctrle.xErr;
			T_HDD.T_Ctrle.xExecute:=FALSE;
			T_HDD.T_Ctrle.xLocked:=FALSE;
			xReadPassword:=FALSE;
		(* error *)
		99:	T_Password.T_Ctrle.xDone:=FALSE;
			T_Password.T_Ctrle.xErr:=TRUE;
			T_Password.T_Ctrle.udiErrorID:=16#F1000 + T_Password.T_Ctrle.iFunction;
			T_HDD.T_Ctrle.xReset:=T_HDD.T_Ctrle.xErr;
			T_HDD.T_Ctrle.xExecute:=FALSE;
			T_HDD.T_Ctrle.xLocked:=FALSE;
			xReadPassword:=FALSE;
		END_CASE;
	END_IF;

(* read Operator Password *)
	IF xWritePassword THEN
		CASE iStepFunction OF
		(* start timeout *)
		1:	TimerFileLocked(IN:=FALSE);
			T_Password.T_Ctrle.udiGetOperatorPassword:=T_Password.T_Ctrle.udiSetOperatorPassword;
			T_Password.T_Ctrle.sGetOperatorPassword:=UDINT_TO_STRING(T_Password.T_Ctrle.udiGetOperatorPassword);
			iStepFunction:=iStepFunction + 1;
		(* Create Password File *)
		2:	IF T_HDD.T_Ctrle.xDone AND NOT(T_HDD.T_Ctrle.xErr) AND NOT(T_HDD.T_Ctrle.xLocked) THEN
				T_HDD.T_Data.sData:=sDeleteData;
				T_HDD.T_Data.sData[1]:=CONCAT(T_Password.T_Ctrle.sGetOperatorPassword,';');	(* Set Password to file *)
				sTmp:=CONCAT(cssRootPLC,'Bore800\Password\OperatorPassword.txt');
				T_HDD.T_File.sPathAndFileName:=sTmp;
				T_HDD.T_Ctrle.iFunction:=2;
				T_HDD.T_Ctrle.xExecute:=TRUE;
				(* next step *)
				iStepFunction:=iStepFunction + 1;
			ELSE
				(* activ error if time out done, HDD not ready *)
				IF TimerFileLocked.Q THEN
					 iStepFunction:=90;
				END_IF
			END_IF;
		(* waiting flag *)
		3:	IF T_HDD.T_Ctrle.xDone AND NOT(T_HDD.T_Ctrle.xErr) THEN iStepFunction:=90; END_IF
			IF T_HDD.T_Ctrle.xErr THEN iStepFunction:=iStepFunction + 1; (* evtl. besteht das Verzeichnis nicht *) END_IF
		(* Create FirstLevel directory *)
		4:	sTmp:=CONCAT(cssRootPLC,'Bore800\');
			(* activ read *)
			T_HDD.T_Ctrle.iFunction:=7;
			T_HDD.T_File.sDirectoryPath:=sTmp;
			T_HDD.T_Ctrle.xExecute:=TRUE;
			(* next step *)
			iStepFunction:=iStepFunction + 1;
		(* waiting flag *)
		5:	IF T_HDD.T_Ctrle.xDone AND NOT(T_HDD.T_Ctrle.xErr) THEN iStepFunction:=iStepFunction + 1; END_IF
			IF T_HDD.T_Ctrle.xErr THEN T_HDD.T_Ctrle.xReset:=TRUE; iStepFunction:=iStepFunction + 1; (* Vielleicht besteht schon dieses Verzeichnis *) END_IF
		(* Create SecondLevel directory *)
		6:	IF NOT(T_HDD.T_Ctrle.xReset) AND T_HDD.T_Ctrle.xDone THEN
				sTmp:=CONCAT(cssRootPLC,'Bore800\Password\');
				(* activ read *)
				T_HDD.T_Ctrle.iFunction:=7;
				T_HDD.T_File.sDirectoryPath:=sTmp;
				T_HDD.T_Ctrle.xExecute:=TRUE;
				(* next step *)
				iStepFunction:=iStepFunction + 1;
			END_IF;
		(* waiting flag *)
		7:	IF T_HDD.T_Ctrle.xDone AND NOT(T_HDD.T_Ctrle.xErr) THEN iStepFunction:=iStepFunction + 1; END_IF
			IF T_HDD.T_Ctrle.xErr THEN T_HDD.T_Ctrle.xReset:=TRUE; iStepFunction:=99; (* generelles Problem mit dem schreiben auf die Flash Karte *) END_IF
		(* Create again Password File *)
		8:	IF T_HDD.T_Ctrle.xDone AND NOT(T_HDD.T_Ctrle.xErr) AND NOT(T_HDD.T_Ctrle.xLocked) THEN
				T_HDD.T_Data.sData:=sDeleteData;
				T_HDD.T_Data.sData[1]:=CONCAT(T_Password.T_Ctrle.sGetOperatorPassword,';');	(* Set Password to file *)
				sTmp:=CONCAT(cssRootPLC,'Bore800\Password\OperatorPassword.txt');
				T_HDD.T_File.sPathAndFileName:=sTmp;
				T_HDD.T_Ctrle.iFunction:=2;
				T_HDD.T_Ctrle.xExecute:=TRUE;
				(* next step *)
				iStepFunction:=iStepFunction + 1;
			ELSE
				(* activ error if time out done, HDD not ready *)
				IF TimerFileLocked.Q THEN
					 iStepFunction:=90;
				END_IF
			END_IF;
		(* waiting flag *)
		9:	IF T_HDD.T_Ctrle.xDone AND NOT(T_HDD.T_Ctrle.xErr) THEN iStepFunction:=90; END_IF
			IF T_HDD.T_Ctrle.xErr THEN iStepFunction:=iStepFunction + 1; (* abbrechen, da schon wieder nicht geschrieben werden konnte *) END_IF
		(* reset error *)
		80:	T_HDD.T_Ctrle.xReset:=TRUE;
			iStepFunction:=91;
		(* done *)
		90:	T_Password.T_Ctrle.xDone:=TRUE;
			T_Password.T_Ctrle.xErr:=FALSE;
			T_Password.T_Ctrle.udiErrorID:=16#0;
			T_HDD.T_Ctrle.xLocked:=FALSE;
			xWritePassword:=FALSE;
		(* start read error *)
		91:	T_Password.T_Ctrle.xDone:=FALSE;
			T_Password.T_Ctrle.xErr:=TRUE;
			T_Password.T_Ctrle.udiErrorID:=16#F1000 + T_Password.T_Ctrle.iFunction;
			T_HDD.T_Ctrle.xReset:=T_HDD.T_Ctrle.xErr;
			T_HDD.T_Ctrle.xExecute:=FALSE;
			T_HDD.T_Ctrle.xLocked:=FALSE;
			xWritePassword:=FALSE;
		(* error *)
		99:	T_Password.T_Ctrle.xDone:=FALSE;
			T_Password.T_Ctrle.xErr:=TRUE;
			T_Password.T_Ctrle.udiErrorID:=16#F1000 + T_Password.T_Ctrle.iFunction;
			T_HDD.T_Ctrle.xReset:=T_HDD.T_Ctrle.xErr;
			T_HDD.T_Ctrle.xExecute:=FALSE;
			T_HDD.T_Ctrle.xLocked:=FALSE;
			xWritePassword:=FALSE;
		END_CASE;
	END_IF;
END_FUNCTION_BLOCK

(* POU GENERAL/PROCESSDATA/FB_PROCESSDATA, ST *)
FUNCTION_BLOCK FB_PROCESSDATA
VAR_INPUT
END_VAR
VAR_IN_OUT
	T_ProcessData:ST_PROCESSDATA;
	T_PartAnalysis:ST_PARTANALYSIS;
	T_HDD:ST_HDD;
END_VAR
VAR_OUTPUT
END_VAR
VAR
	sTmp:STRING(255);
	RisingEdgeReset:R_TRIG;
	RisingEdgeExecute:R_TRIG;
	xConfirmResetFB: BOOL;
	TimerFileLocked:TON;
	tTimeOut: TIME;
	iStepFunction: INT;
	xTmp: BOOL;
	TimerOut: TON;
	FBNT_GetTime:NT_GetTime;
	sGetDate: STRING;
	xInit: BOOL;
	sDeleteData: ARRAY[1..csiMaxFileLine] OF STRING(csiMaxCharPerLine);
	iStepFunction_Intern: INT;
	iStepFunction_Check: INT;
	xWriteData: BOOL;
	sYear: STRING;
	sMonth: STRING;
	sDay: STRING;
	sHour: STRING;
	sMinute: STRING;
	sSecond: STRING;
	xReadTimeStamp: BOOL;
	iStep_TimeStamp: INT;
	iStepCountWriteDirectory: INT;
	xWriteFileFirstTime: BOOL;
	ii: INT;
	sWorkPartQuality: STRING;
	sFirstHC: STRING;
	sHCCounter: STRING;
	sHCCounterCentering: STRING;
	sHCCounterTorque: STRING;
	sHCCounterSpeed:STRING;	(* IGS *)
	sCycleTime: STRING;
	sWorkTime: STRING;
	sInfeedCounterZ: STRING;
	iDataPointer: INT;
	sNumberHole: STRING;
END_VAR
(****************************************************************************************************************************************************)
(***********                                               This Functionblock manage the FTP Client upload file                                                        ************)
(****************************************************************************************************************************************************)
(* waiting for reset *)
	RisingEdgeReset(CLK:=T_ProcessData.T_Ctrle.xReset);
	IF RisingEdgeReset.Q THEN
	(* init. structure *)
		T_ProcessData.T_Ctrle.xExecute:=FALSE;
		T_ProcessData.T_Ctrle.xReset:=FALSE;
		T_ProcessData.T_Ctrle.xDone:=FALSE;
		T_ProcessData.T_Ctrle.xErr:=FALSE;
		T_ProcessData.T_Ctrle.udiErrorID:=0;
		T_ProcessData.T_Ctrle.iFunction:=0;
		IF T_HDD.T_Ctrle.xErr THEN T_HDD.T_Ctrle.xReset:=TRUE; END_IF
		T_HDD.T_Ctrle.xLocked:=FALSE;
		(* Reset HDD if error activ *)
		(* Init. variable *)
		xWriteData:=FALSE;
		(* set flag done *)
		xConfirmResetFB:=TRUE;
		(* exit function *)
		RETURN;
	ELSE
		IF xConfirmResetFB THEN
		(* confirm reset FB *)
			T_ProcessData.T_Ctrle.xDone:=TRUE;
			T_ProcessData.T_Ctrle.xErr:=FALSE;
			T_ProcessData.T_Ctrle.udiErrorID:=0;
			T_ProcessData.T_Ctrle.iFunction:=0;
			(* init. variable *)
			xConfirmResetFB:=FALSE;
		END_IF
	END_IF

TimerFileLocked(IN:=TRUE, PT:=T#10S);

(* waiting for execute *)
	RisingEdgeExecute(CLK:=T_ProcessData.T_Ctrle.xExecute);
	IF RisingEdgeExecute.Q THEN
		T_ProcessData.T_Ctrle.xExecute:=FALSE;
		CASE T_ProcessData.T_Ctrle.iFunction OF
		(* Write Data File on USB Stick *)
		1:	xWriteData:=TRUE;
			tTimeOut:=T#300s;
		ELSE
		(* function not implemented *)
			 T_ProcessData.T_Ctrle.xDone:=FALSE;
			 T_ProcessData.T_Ctrle.xErr:=TRUE;
			 T_ProcessData.T_Ctrle.udiErrorID:=200;
			 (* exit FB *)
			 RETURN;
		END_CASE
		(* Init. variable *)
		T_ProcessData.T_Ctrle.xDone:=FALSE;
		T_ProcessData.T_Ctrle.xErr:=FALSE;
		T_ProcessData.T_Ctrle.udiErrorID:=16#0;
		(* init. step *)
		iStepFunction:=1;
		iStepFunction_Intern:=1;
		iStepFunction_Check:=1;
		RETURN;
	END_IF

(* Monitor time out *)
	xTmp:=	NOT T_ProcessData.T_Ctrle.xDone
			AND NOT T_ProcessData.T_Ctrle.xErr;
	TimerOut(IN:=xTmp, PT:=tTimeOut);
	IF TimerOut.Q THEN iStepFunction:=97; END_IF

(* Read or Write profile *)
	IF xWriteData THEN
		CASE iStepFunction OF
		(* check if HDD state *)
		(* start timeout *)
		1:	TimerFileLocked(IN:=FALSE);
			iStepFunction:=iStepFunction + 1;
			iStepCountWriteDirectory:=0;
			xWriteFileFirstTime:=FALSE;
		(* file name and activ read or write *)
		2:	IF T_HDD.T_Ctrle.xDone AND NOT(T_HDD.T_Ctrle.xErr) AND NOT(T_HDD.T_Ctrle.xLocked) THEN
				T_HDD.T_Ctrle.xLocked:=TRUE;
				(* next step *)
				iStepFunction:=iStepFunction + 1;
				T_HDD.T_Data.sData:=sDeleteData;
			ELSE
				(* activ error if time out done, HDD not ready *)
				IF TimerFileLocked.Q THEN
					 iStepFunction:=91;
				END_IF
			END_IF;
		(* Überprüfe zuerst welche USB Stick als ProcessData definiert ist *)
		3:	IF (gsDriveNameProcessData = '') THEN
				IF NOT(gxHardwareOFF) THEN
					sTmp:='D:\PROCESSDATA.txt';
				ELSE
					sTmp:='C:\PROCESSDATA.txt';
					(*sTmp:='\Hard Disk2\PROCESSDATA.txt';*)
				END_IF;
				T_HDD.T_File.sPathAndFileName:=sTmp;
				T_HDD.T_Ctrle.iFunction:=1;
				T_HDD.T_Ctrle.xExecute:=TRUE;
				(* next step *)
				iStepFunction:=iStepFunction + 1;
			ELSE
				(* next step *)
				iStepFunction:=iStepFunction + 4;
			END_IF;
		(* waiting flag *)
		4:	IF T_HDD.T_Ctrle.xDone AND NOT(T_HDD.T_Ctrle.xErr) THEN
				iStepFunction:=iStepFunction + 3;
				IF NOT(gxHardwareOFF) THEN
					gsDriveNameProcessData:='D:\';
				ELSE
					gsDriveNameProcessData:='C:\';
					(*gsDriveNameProcessData:='\Hard Disk2\';*)
				END_IF;
			END_IF
			IF T_HDD.T_Ctrle.xErr THEN T_HDD.T_Ctrle.xReset:=TRUE; iStepFunction:=iStepFunction + 1; END_IF
		5:	IF T_HDD.T_Ctrle.xDone AND NOT(T_HDD.T_Ctrle.xErr) AND NOT(T_HDD.T_Ctrle.xLocked) THEN
				T_HDD.T_Ctrle.xLocked:=TRUE;
				IF NOT(gxHardwareOFF) THEN
					sTmp:='E:\PROCESSDATA.txt';
				ELSE
					sTmp:='C:\PROCESSDATA.txt';
					(*sTmp:='\Hard Disk2\PROCESSDATA.txt';*)
				END_IF;
				T_HDD.T_File.sPathAndFileName:=sTmp;
				T_HDD.T_Ctrle.iFunction:=1;
				T_HDD.T_Ctrle.xExecute:=TRUE;
				(* next step *)
				iStepFunction:=iStepFunction + 1;
			END_IF;
		(* waiting flag *)
		6:	IF T_HDD.T_Ctrle.xDone AND NOT(T_HDD.T_Ctrle.xErr) THEN iStepFunction:=iStepFunction + 1; gsDriveNameProcessData:='E:\'; END_IF
			IF T_HDD.T_Ctrle.xErr THEN T_HDD.T_Ctrle.xReset:=TRUE; iStepFunction:=99; END_IF
		7:	IF NOT(xReadTimeStamp) THEN
				xReadTimeStamp:=TRUE;	(* Zeitstempel lesen *)
				iStepFunction:=iStepFunction + 1;
			END_IF;
		8:	IF NOT(xReadTimeStamp) THEN
				sGetDate:=sYear;
				sGetDate:=CONCAT(sGetDate,'-');
				sGetDate:=CONCAT(sGetDate,sMonth);
				sGetDate:=CONCAT(sGetDate,'-');
				sGetDate:=CONCAT(sGetDate,sDay);
				sGetDate:=CONCAT(sGetDate,'_');
				sGetDate:=CONCAT(sGetDate,sHour);
				sGetDate:=CONCAT(sGetDate,'-');
				sGetDate:=CONCAT(sGetDate,sMinute);
				sGetDate:=CONCAT(sGetDate,'-');
				sGetDate:=CONCAT(sGetDate,sSecond);
				IF (T_PartAnalysis.sFileName = '') THEN
					xWriteFileFirstTime:=TRUE;
					T_PartAnalysis.sFileName:=CONCAT(sGetDate,'-St');
					T_PartAnalysis.sFileName:=CONCAT(T_PartAnalysis.sFileName,UINT_TO_STRING(gciStationSt1));
					T_PartAnalysis.sFileName:=CONCAT(T_PartAnalysis.sFileName,'.csv');
				END_IF;
				iStepFunction:=iStepFunction + 1;
			END_IF;
			xInit:=FALSE;
		(* file name and activ read or write *)
		9:	(* activ write *)
			IF T_HDD.T_Ctrle.xDone AND NOT(T_HDD.T_Ctrle.xErr) THEN
				T_HDD.T_Data.sData:=sDeleteData;
				(* copy profile to HDD data structure *)
				 iStepFunction:=iStepFunction + 1;
				(* next step *)
			END_IF;
		(* activ write *)
		10:	sTmp:=CONCAT(gsDriveNameProcessData,'PROCESSDATA\');
			sTmp:=CONCAT(sTmp,T_PartAnalysis.sFileName);
			T_HDD.T_File.sPathAndFileName:=sTmp;
			iDataPointer:=1;
			IF xWriteFileFirstTime THEN
				(*T_HDD.T_Data.sData[iDataPointer]:='WPNumber;Timestamp;Hole Quality;FirstHC(mm);HC Counter(D);HC Counter(T);Cycle time(s);Work time(s);Z Inf.Counter;';*)	(* alt *)
				T_HDD.T_Data.sData[iDataPointer]:='WstkNr;Zeitstempel;Loch Qualität;ErsterHC(mm);HC Zähler(A);HC Zähler(D);HC Zähler(G);Zyklus(s);Bearb(s);Z Einf.Zähler;HC Zähler(Zentr.);';		(* IGS *)
				iDataPointer:=iDataPointer + 1;
			END_IF;
			FOR ii:=1 TO ciMaxWP DO
				IF (T_PartAnalysis.adiNumberHole[ii] = T_NovRam.T_Parameter.T_PartAnalysis[gciStationSt1].diActual_NumberHoleToWork) THEN
					sNumberHole:=DINT_TO_STRING(T_PartAnalysis.adiNumberHole[ii]);
					sGetDate:=sYear;
					sGetDate:=CONCAT(sGetDate,'.');
					sGetDate:=CONCAT(sGetDate,sMonth);
					sGetDate:=CONCAT(sGetDate,'.');
					sGetDate:=CONCAT(sGetDate,sDay);
					sGetDate:=CONCAT(sGetDate,' ');
					sGetDate:=CONCAT(sGetDate,sHour);
					sGetDate:=CONCAT(sGetDate,':');
					sGetDate:=CONCAT(sGetDate,sMinute);
					sGetDate:=CONCAT(sGetDate,':');
					sGetDate:=CONCAT(sGetDate,sSecond);
					CASE T_PartAnalysis.abWorkPartQuality[ii] OF
					0:	sWorkPartQuality:='Hole not worked';
					1:	sWorkPartQuality:='Go HC';
					2:	sWorkPartQuality:='Go No HC';
					3:	sWorkPartQuality:='NoGo minTime';
					4:	sWorkPartQuality:='NoGo maxTime';
					5:	sWorkPartQuality:='NoGo insert fail';
					6:	sWorkPartQuality:='NoGo NoWP';
					7:	sWorkPartQuality:='Working';
					8:	sWorkPartQuality:='Cycle aborted';
					10:	sWorkPartQuality:='NoGo HC Centr.';
					END_CASE;
					sFirstHC:=REAL_TO_STRING(T_PartAnalysis.arFirstHC[ii]);
					sHCCounter:=INT_TO_STRING(T_PartAnalysis.aiHCCounter[ii]);
					sHCCounterCentering:=INT_TO_STRING(T_PartAnalysis.aiHCCounterCentering[ii]);
					sHCCounterTorque:=INT_TO_STRING(T_PartAnalysis.aiHCCounterTorque[ii]);
					sHCCounterSpeed:=INT_TO_STRING(T_PartAnalysis.aiHCCounterSpeed[ii]);
					sCycleTime:=REAL_TO_STRING(DINT_TO_REAL(T_PartAnalysis.adiCycleTime[ii]) / 1000.0);
					sWorkTime:=REAL_TO_STRING(DINT_TO_REAL(T_PartAnalysis.adiWorkTime[ii]) / 1000.0);
					sInfeedCounterZ:=BYTE_TO_STRING(T_PartAnalysis.abInfeedCounterZ[ii]);
					T_HDD.T_Data.sData[iDataPointer]:=CONCAT(sNumberHole,';');
					T_HDD.T_Data.sData[iDataPointer]:=CONCAT(T_HDD.T_Data.sData[iDataPointer],sGetDate);
					T_HDD.T_Data.sData[iDataPointer]:=CONCAT(T_HDD.T_Data.sData[iDataPointer],';');
					T_HDD.T_Data.sData[iDataPointer]:=CONCAT(T_HDD.T_Data.sData[iDataPointer],sWorkPartQuality);
					T_HDD.T_Data.sData[iDataPointer]:=CONCAT(T_HDD.T_Data.sData[iDataPointer],';');
					T_HDD.T_Data.sData[iDataPointer]:=CONCAT(T_HDD.T_Data.sData[iDataPointer],sFirstHC);
					T_HDD.T_Data.sData[iDataPointer]:=CONCAT(T_HDD.T_Data.sData[iDataPointer],';');
					T_HDD.T_Data.sData[iDataPointer]:=CONCAT(T_HDD.T_Data.sData[iDataPointer],sHCCounter);
					T_HDD.T_Data.sData[iDataPointer]:=CONCAT(T_HDD.T_Data.sData[iDataPointer],';');
					T_HDD.T_Data.sData[iDataPointer]:=CONCAT(T_HDD.T_Data.sData[iDataPointer],sHCCounterTorque);
					T_HDD.T_Data.sData[iDataPointer]:=CONCAT(T_HDD.T_Data.sData[iDataPointer],';');
					T_HDD.T_Data.sData[iDataPointer]:=CONCAT(T_HDD.T_Data.sData[iDataPointer],sHCCounterSpeed);
					T_HDD.T_Data.sData[iDataPointer]:=CONCAT(T_HDD.T_Data.sData[iDataPointer],';');
					T_HDD.T_Data.sData[iDataPointer]:=CONCAT(T_HDD.T_Data.sData[iDataPointer],sCycleTime);
					T_HDD.T_Data.sData[iDataPointer]:=CONCAT(T_HDD.T_Data.sData[iDataPointer],';');
					T_HDD.T_Data.sData[iDataPointer]:=CONCAT(T_HDD.T_Data.sData[iDataPointer],sWorkTime);
					T_HDD.T_Data.sData[iDataPointer]:=CONCAT(T_HDD.T_Data.sData[iDataPointer],';');
					T_HDD.T_Data.sData[iDataPointer]:=CONCAT(T_HDD.T_Data.sData[iDataPointer],sInfeedCounterZ);
					T_HDD.T_Data.sData[iDataPointer]:=CONCAT(T_HDD.T_Data.sData[iDataPointer],';');
					T_HDD.T_Data.sData[iDataPointer]:=CONCAT(T_HDD.T_Data.sData[iDataPointer],sHCCounterCentering);
					T_HDD.T_Data.sData[iDataPointer]:=CONCAT(T_HDD.T_Data.sData[iDataPointer],';');
				END_IF;
			END_FOR;
			T_HDD.T_Ctrle.iFunction:=3;
			T_HDD.T_Ctrle.xExecute:=TRUE;
			(* next step *)
			iStepFunction:=iStepFunction + 1;
		(* waiting flag *)
		11:	IF T_HDD.T_Ctrle.xDone AND NOT(T_HDD.T_Ctrle.xErr) THEN iStepFunction:=90; END_IF
			IF T_HDD.T_Ctrle.xErr THEN T_HDD.T_Ctrle.xReset:=TRUE; iStepFunction:=iStepFunction + 1; iStepCountWriteDirectory:=iStepCountWriteDirectory + 1; END_IF
		(* Create Directory *)
		12:	IF T_HDD.T_Ctrle.xDone AND NOT(T_HDD.T_Ctrle.xErr) THEN
				IF (iStepCountWriteDirectory < 2) THEN
					sTmp:=CONCAT(gsDriveNameProcessData,'PROCESSDATA\');
					T_HDD.T_Ctrle.iFunction:=7;
					T_HDD.T_File.sDirectoryPath:=sTmp;
					T_HDD.T_Ctrle.xExecute:=TRUE;
					(* next step *)
					iStepFunction:=iStepFunction + 1;
				ELSE
					iStepFunction:=98;
				END_IF;
			END_IF;
		(* waiting flag *)
		13:	IF T_HDD.T_Ctrle.xDone AND NOT(T_HDD.T_Ctrle.xErr) THEN iStepFunction:=10; END_IF
			IF T_HDD.T_Ctrle.xErr THEN T_HDD.T_Ctrle.xReset:=TRUE; iStepFunction:=98; END_IF
		(* done *)
		90:	T_ProcessData.T_Ctrle.xDone:=TRUE;
			T_ProcessData.T_Ctrle.xErr:=FALSE;
			T_ProcessData.T_Ctrle.udiErrorID:=16#0;
			T_HDD.T_Ctrle.xExecute:=FALSE;
			T_HDD.T_Ctrle.xLocked:=FALSE;
			xWriteData:=FALSE;
		(* start read error *)
		91:	T_ProcessData.T_Ctrle.xDone:=FALSE;
			T_ProcessData.T_Ctrle.xErr:=TRUE;
			T_ProcessData.T_Ctrle.udiErrorID:=201;	(* HDD steht nicht Bereit *)
			T_HDD.T_Ctrle.xReset:=T_HDD.T_Ctrle.xErr;
			T_HDD.T_Ctrle.xExecute:=FALSE;
			T_HDD.T_Ctrle.xLocked:=FALSE;
			xWriteData:=FALSE;
		(* error *)
		97:	T_ProcessData.T_Ctrle.xDone:=FALSE;
			T_ProcessData.T_Ctrle.xErr:=TRUE;
			T_ProcessData.T_Ctrle.udiErrorID:=202;	(* Timeout beim Schreiben auf USB-Stick *)
			T_HDD.T_Ctrle.xReset:=T_HDD.T_Ctrle.xErr;
			T_HDD.T_Ctrle.xExecute:=FALSE;
			T_HDD.T_Ctrle.xLocked:=FALSE;
			xWriteData:=FALSE;
			gsDriveNameProcessData:='';
		(* error *)
		98:	T_ProcessData.T_Ctrle.xDone:=FALSE;
			T_ProcessData.T_Ctrle.xErr:=TRUE;
			T_ProcessData.T_Ctrle.udiErrorID:=203;	(* USB Stick nicht schreibbar *)
			T_HDD.T_Ctrle.xReset:=T_HDD.T_Ctrle.xErr;
			T_HDD.T_Ctrle.xExecute:=FALSE;
			T_HDD.T_Ctrle.xLocked:=FALSE;
			xWriteData:=FALSE;
			gsDriveNameProcessData:='';
		(* error *)
		99:	T_ProcessData.T_Ctrle.xDone:=FALSE;
			T_ProcessData.T_Ctrle.xErr:=TRUE;
			T_ProcessData.T_Ctrle.udiErrorID:=204;	(* USB Stick nicht gefunden *)
			T_HDD.T_Ctrle.xReset:=T_HDD.T_Ctrle.xErr;
			T_HDD.T_Ctrle.xExecute:=FALSE;
			T_HDD.T_Ctrle.xLocked:=FALSE;
			xWriteData:=FALSE;
			gsDriveNameProcessData:='';
		END_CASE
	END_IF

(* Zeitstempel lesen *)
	IF xReadTimeStamp THEN
		CASE iStep_TimeStamp OF
		1:	FBNT_GetTime(	NETID:= '',
							START:=FALSE );
			iStep_TimeStamp:=iStep_TimeStamp + 1;
		2:	FBNT_GetTime(	NETID:= '',
							START:= TRUE,
							TMOUT:= T#2s);
			IF NOT(FBNT_GetTime.BUSY) OR FBNT_GetTime.ERR THEN
				IF NOT(FBNT_GetTime.ERR) THEN
					sYear:=WORD_TO_STRING(FBNT_GetTime.TIMESTR.wYear);
					IF (FBNT_GetTime.TIMESTR.wMonth < 10) THEN
						sMonth:=CONCAT('0',WORD_TO_STRING(FBNT_GetTime.TIMESTR.wMonth));
					ELSE
						sMonth:=WORD_TO_STRING(FBNT_GetTime.TIMESTR.wMonth);
					END_IF;
					IF (FBNT_GetTime.TIMESTR.wDay < 10) THEN
						sDay:=CONCAT('0',WORD_TO_STRING(FBNT_GetTime.TIMESTR.wDay));
					ELSE
						sDay:=WORD_TO_STRING(FBNT_GetTime.TIMESTR.wDay);
					END_IF;
					IF (FBNT_GetTime.TIMESTR.wHour < 10) THEN
						sHour:=CONCAT('0',WORD_TO_STRING(FBNT_GetTime.TIMESTR.wHour));
					ELSE
						sHour:=WORD_TO_STRING(FBNT_GetTime.TIMESTR.wHour);
					END_IF;
					IF (FBNT_GetTime.TIMESTR.wMinute < 10) THEN
						sMinute:=CONCAT('0',WORD_TO_STRING(FBNT_GetTime.TIMESTR.wMinute));
					ELSE
						sMinute:=WORD_TO_STRING(FBNT_GetTime.TIMESTR.wMinute);
					END_IF;
					IF (FBNT_GetTime.TIMESTR.wSecond < 10) THEN
						sSecond:=CONCAT('0',WORD_TO_STRING(FBNT_GetTime.TIMESTR.wSecond));
					ELSE
						sSecond:=WORD_TO_STRING(FBNT_GetTime.TIMESTR.wSecond);
					END_IF;
				ELSE
					(* Fehler beim lesen der Systemzeit, daher wird ein default-Wert gesetzt *)
					sYear:='0000';
					sMonth:='00';
					sDay:='00';
					sHour:='00';
					sMinute:='00';
					sSecond:='00';
				END_IF;
				FBNT_GetTime(	NETID:= '',
								START:=FALSE );
				xReadTimeStamp:=FALSE;
			END_IF;
		END_CASE;
	ELSE
		iStep_TimeStamp:=1;
	END_IF;
END_FUNCTION_BLOCK

(* POU GENERAL/FB_ControlLamp, ST *)
FUNCTION_BLOCK FB_ControlLamp
VAR_INPUT
	xStartUpCompleted:BOOL;
	iStateMessage:INT;
	xSetupActive:BOOL;
	xPreWarningActive:BOOL;
END_VAR
VAR_IN_OUT
	TProcess : ST_PROCESS;
	TCtrlePanel:ST_CTRLEPANEL;
END_VAR
VAR_OUTPUT
	xLampGreen:BOOL;
	xLampRed:BOOL;
	xLampYellow:BOOL;
END_VAR
VAR
(* Timer *)
	TimerON:TON;
	TimerOFF:TOF;
	tTimerCadence:TIME;
	xTimerSignal:BOOL;
(* variable *)
	xFirstExecution:BOOL;
	xPanelLedBlinked: BOOL;
(* Tmp *)
	xTmp:BOOL;
	bLampGreen: BYTE;
	bLampYellow: BYTE;
	bLampRed: BYTE;
END_VAR
(* First execution *)
	IF NOT xFirstExecution THEN
		(* Init. variable *)
		tTimerCadence:=T#0.5s;
		xTimerSignal:=FALSE;
		(* Timer *)
		TimerON(IN:=FALSE);
		TimerOFF(IN:=TRUE);
		(* Confirm execution *)
		xFirstExecution:=TRUE;
	END_IF

(* Each cycle, init. lamp state *)
	xLampGreen:=FALSE;
	xLampRed:=FALSE;
	xLampYellow:=FALSE;
	TCtrlePanel.udiLED:=16#0;

(* Each cycle, init. lamp state function *)
	xTmp:=FALSE;
	bLampGreen:=0;bLampYellow:=0;bLampRed:=0;
	xPanelLedBlinked:=FALSE;

	IF NOT(xStartUpCompleted) THEN
		(* Maschine ist eingeschaltet, Betriebssystem ist geladen resp. SPS steht bereit, Maschine wurde aber noch nicht aufgestartet oder ist noch am aufstarten *)
		bLampGreen:=1;bLampYellow:=1;bLampRed:=1;	(* Grün ON, Gelb ON, Rot ON *)
	ELSE
		IF (iStateMessage = 401) THEN
			(* Error state *)
			(* Automatik- oder Einrichtbetrieb-->Störung (Warnung aber nicht Aktiv) *)
			bLampGreen:=0;bLampYellow:=0;bLampRed:=1;	(* Grün OFF, Gelb OFF, Rot ON *)
			xPanelLedBlinked:=TRUE;
		ELSIF NOT(TProcess.T_Ctrle.xDone)  AND NOT(xSetupActive) THEN
			IF NOT(xPreWarningActive) THEN
				(* Automatikbetrieb --> Prozess (Automatik, Masch.Ref, WstkEntladen) Aktiv *)
				bLampGreen:=1;bLampYellow:=0;bLampRed:=0;	(* Grün ON, Gelb OFF, Rot OFF *)
			ELSE
				(* Automatikbetrieb --> Prozess Aktiv --> Vorwarnung Materialmangel (Wstk, Wz, Kühlmittelfüllstand) *)
				bLampGreen:=1;bLampYellow:=1;bLampRed:=0;	(* Grün ON, Gelb ON, Rot OFF *)
			END_IF;
		ELSIF TProcess.T_Ctrle.xDone AND NOT(xSetupActive) THEN
			(* Automatikbetrieb --> Maschinenstillstand ohne Störung *)
			IF NOT(xPreWarningActive) THEN
				bLampGreen:=2;bLampYellow:=0;bLampRed:=0;	(* Grün BLINK, Gelb OFF, Rot OFF *)
			ELSE
				bLampGreen:=2;bLampYellow:=1;bLampRed:=0;	(* Grün BLINK, Gelb ON, Rot OFF *)
			END_IF;
		ELSIF xSetupActive THEN
			(* Einrichtbetrieb --> unabhängig ob eine Bewegung stattfindet oder nicht *)
			bLampGreen:=2;bLampYellow:=2;bLampRed:=2;	(* Grün BLINK, Gelb BLINK, Rot BLINK *)
		ELSE
			(* Maschine ist ausgeschaltet oder Maschine ist eingeschaltet, aber Betriebssystem ist noch nicht geladen resp. SPS steht noch nicht bereit *)
			bLampGreen:=0;bLampYellow:=0;bLampRed:=0;	(* Grün OFF, Gelb OFF, Rot OFF *)
		END_IF;
	END_IF;

(* Blink *)
	TimerON(IN:=TRUE,PT:=tTimerCadence);
	IF TimerON.Q THEN
		TimerOFF(IN:=FALSE,PT:=tTimerCadence);
		IF NOT TimerOFF.Q THEN TimerON(IN:=FALSE); TimerOFF(IN:=TRUE); END_IF
	END_IF
(* Grüne Lampe-->Werkerruflampe *)
	IF (bLampGreen = 0) THEN
		xLampGreen:=FALSE;	(* Grüne Lampe ausgeschaltet *)
	ELSIF (bLampGreen = 1) THEN
		xLampGreen:=TRUE;	(* Grüne Lampe eingeschaltet *)
	ELSIF (bLampGreen = 2) THEN
		xLampGreen:=TimerON.Q;	(* Grüne Lampe blinkt *)
	END_IF;
(* Gelbe Lampe-->Werkerruflampe *)
	IF (bLampYellow = 0) THEN
		xLampYellow:=FALSE;	(* Gelbe Lampe ausgeschaltet *)
	ELSIF (bLampYellow = 1) THEN
		xLampYellow:=TRUE;	(* Gelbe Lampe eingeschaltet *)
	ELSIF (bLampYellow = 2) THEN
		xLampYellow:=TimerON.Q;	(* Gelbe Lampe blinkt *)
	END_IF;
(* Rote Lampe-->Werkerruflampe *)
	IF (bLampRed = 0) THEN
		xLampRed:=FALSE;	(* Rote Lampe ausgeschaltet *)
	ELSIF (bLampRed = 1) THEN
		xLampRed:=TRUE;	(* Rote Lampe eingeschaltet *)
	ELSIF (bLampRed = 2) THEN
		xLampRed:=TimerON.Q;	(* Rote Lampe blinkt *)
	END_IF;

(* Panel led blinked *)
	IF xPanelLedBlinked THEN
		IF TimerON.Q THEN TCtrlePanel.udiLED:=16#3FF; ELSE TCtrlePanel.udiLED:=16#0; END_IF
	END_IF
END_FUNCTION_BLOCK

(* POU PRG_USB_IO_PANEL, ST *)
PROGRAM PRG_USB_IO_PANEL
VAR
(* Panel tastatur *)
	(* function bloc *)
	fbCtrlePanel_IO:FBHW_PANEL_IO;
	(* IO connection *)

	IarxCtrlePanelButton AT %I* : ARRAY[1..10] OF BOOL;
	QarxCtrlePanelLed AT %Q* : ARRAY[1..10] OF BOOL;
END_VAR
(* Call FB *)
	fbCtrlePanel_IO(	arxButton:=IarxCtrlePanelButton,
					T_CtrlePanel:=T_CtrlePanel,
					arxLed=>QarxCtrlePanelLed);
END_PROGRAM

(* POU FB_HARDWARE/FBHW_PANEL_IO, ST *)
FUNCTION_BLOCK FBHW_PANEL_IO
VAR_INPUT
	arxButton:ARRAY[1..10] OF BOOL;
END_VAR
VAR_OUTPUT
	arxLed:ARRAY[1..10] OF BOOL;
END_VAR
VAR_IN_OUT
	T_CtrlePanel:ST_CTRLEPANEL;
END_VAR
VAR
(* variable *)
	xConfirmResetFB:BOOL;
	xConfirmFct:BOOL;
	i: INT;
	si: SINT;
(* trigger *)
	RisingEdgeExecute:R_TRIG;
	RisingEdgeReset:R_TRIG;
END_VAR
(* reset function bloc *)
	RisingEdgeReset(CLK:=T_CtrlePanel.xReset);
	IF RisingEdgeReset.Q THEN
	(* reset output *)
		FOR i := 1 TO 10 DO
			arxLed[i]:=FALSE;
		END_FOR
	(* init. structure *)
		T_CtrlePanel.iFunction:=0;
		T_CtrlePanel.xDone:=FALSE;
		T_CtrlePanel.xErr:=FALSE;
		T_CtrlePanel.udiErrorID:=0;
		T_CtrlePanel.udiButton:=0;
		T_CtrlePanel.udiLED:=0;
	(* confirm reset *)
		xConfirmResetFB:=TRUE;
	(* exit fb *)
		RETURN;
	ELSE
		IF xConfirmResetFB THEN
		(* confirm reset FB *)
			T_CtrlePanel.xDone:=TRUE;
			T_CtrlePanel.xErr:=FALSE;
			T_CtrlePanel.udiErrorID:=0;
			(* Init. variable *)
			xConfirmResetFB:=FALSE;
		END_IF
	END_IF

(* Switch on/off the Led from the control panel *)
	RisingEdgeExecute(CLK:=T_CtrlePanel.xExecute);
	IF RisingEdgeExecute.Q THEN
		CASE T_CtrlePanel.iFunction OF
		(* switch off a specific LED off *)
		-10..-1:	IF arxLed[ABS(T_CtrlePanel.iFunction)] THEN
					arxLed[ABS(T_CtrlePanel.iFunction)]:=FALSE;
					T_CtrlePanel.udiLED:=T_CtrlePanel.udiLED - MUX(ABS(T_CtrlePanel.iFunction)-1,1,2,4,8,16,32,64,128,256,512);
				END_IF
		(* switch off all the LED *)
		0:	FOR i := 1 TO 10 DO
				arxLed[i]:=FALSE;
			END_FOR
			T_CtrlePanel.udiLED:=0;
		(* switch on a specific Led on *)
		1..10:	IF NOT(arxLed[T_CtrlePanel.iFunction]) THEN
					arxLed[T_CtrlePanel.iFunction]:=TRUE;
					T_CtrlePanel.udiLED:=T_CtrlePanel.udiLED + MUX(T_CtrlePanel.iFunction-1,1,2,4,8,16,32,64,128,256,512);
				END_IF
		ELSE
			(* function not implemented *)
			T_CtrlePanel.xDone:=FALSE;
			T_CtrlePanel.xErr:=TRUE;
			T_CtrlePanel.udiErrorID:=16#F000;
			(* exit FB *)
			RETURN;
		END_CASE
		(* Init. variable *)
		T_CtrlePanel.xDone:=FALSE;
		T_CtrlePanel.xErr:=FALSE;
		T_CtrlePanel.udiErrorID:=16#0;
		(* activ confirm *)
		xConfirmFct:=TRUE;
		(* exit FB *)
		RETURN;
	END_IF

(* return the button state *)
	T_CtrlePanel.udiButton:=0;
	FOR i := 0 TO 9 DO
		IF arxButton[i+1] THEN
			T_CtrlePanel.udiButton:=T_CtrlePanel.udiButton + MUX(i,1,2,4,8,16,32,64,128,256,512);
		END_IF
	END_FOR

(* set the led state *)
	FOR si := 0 TO 9 DO
		IF GETBIT32(T_CtrlePanel.udiLED,si) <> 16#0 THEN
			arxLed[si+1]:=TRUE; ELSE arxLed[si+1]:=FALSE; END_IF
	END_FOR

(* wait to confirm *)
	IF xConfirmFct THEN
		T_CtrlePanel.xDone:=TRUE;
		T_CtrlePanel.xErr:=FALSE;
		T_CtrlePanel.udiErrorID:=16#0;
		(* reset variable *)
		xConfirmFct:=FALSE;
	END_IF
END_FUNCTION_BLOCK

(* POU GENERAL/PROFILE/xFctSetOnlineChangeMaxMin, ST *)
FUNCTION xFctSetOnlineChangeMaxMin : BOOL
VAR_INPUT
	ptrProfileOnlineChange:POINTER TO ST_PROFILEONLINECHANGE;
	rMaxToolSpindleSpeed:REAL;
	rMaxForceDeflection:REAL;
	rMaxTorqueLevel:REAL;
	rMinTorqueLevel:REAL;
END_VAR
VAR
END_VAR
(* Init. function state *)
	xFctSetOnlineChangeMaxMin:=FALSE;

(* Set Max/Min for the online change value *)
		ptrProfileOnlineChange^.T_Max.rWorkingOffsetBackward:=0.0;
		ptrProfileOnlineChange^.T_Min.rWorkingOffsetBackward:=-100.0;
		ptrProfileOnlineChange^.T_Max.rWorkingSpeedForward:=150.0;
		ptrProfileOnlineChange^.T_Min.rWorkingSpeedForward:=0.1;
		ptrProfileOnlineChange^.T_Max.rWorkingSpeedBackward:=250.0;
		ptrProfileOnlineChange^.T_Min.rWorkingSpeedBackward:=0.1;
		ptrProfileOnlineChange^.T_Max.rWorkingSpindleSpeed:=rMaxToolSpindleSpeed;
		ptrProfileOnlineChange^.T_Min.rWorkingSpindleSpeed:=rMaxToolSpindleSpeed * -1.0;
		ptrProfileOnlineChange^.T_Max.rForceDeflection:=rMaxForceDeflection;
		ptrProfileOnlineChange^.T_Min.rForceDeflection:=0.1;
		ptrProfileOnlineChange^.T_Max.rTorqueLevelHC:=rMaxTorqueLevel;
		ptrProfileOnlineChange^.T_Min.rTorqueLevelHC:=rMinTorqueLevel;

(* Confirm function execution *)
	xFctSetOnlineChangeMaxMin:=TRUE;
END_FUNCTION

(* POU GENERAL/PROFILE/xFctUpdateOnlineChangeValue, ST *)
FUNCTION xFctUpdateOnlineChangeValue : BOOL
VAR_INPUT
	ptrProfileOnlineChange:POINTER TO ST_PROFILEONLINECHANGE;	(* Min Max Werte der OnlineChange Parameter *)
	ptrProfileOnlineChangeLoad:POINTER TO ST_PROFILEONLINECHANGE_DATA;	(* Min Max Werte der OnlineChange Parameter *)
	ptrExchgParamStationCommon:POINTER TO ST_EXCHG_PARAM_ONLINECHANGE;
	TOnlineChangeParameter:ST_PROFILEONLINECHANGE_DATA;	(* Datenübergabe *)
END_VAR
VAR
(* Tmp variable *)
	rTmp:REAL;
END_VAR
(* Update online value *)
	ptrExchgParamStationCommon^.T_Data:=TOnlineChangeParameter;

(* Update Abs perzent *)
	IF ptrProfileOnlineChange^.T_Min.rWorkingOffsetBackward <> 0 THEN
		ptrExchgParamStationCommon^.T_DataValPercentAbs.rWorkingOffsetBackward
			:=ABS(TOnlineChangeParameter.rWorkingOffsetBackward/ptrProfileOnlineChange^.T_Min.rWorkingOffsetBackward*100);
	ELSE ptrExchgParamStationCommon^.T_DataValPercentAbs.rWorkingOffsetBackward:=-1; END_IF
	IF ptrProfileOnlineChange^.T_Max.rWorkingSpeedForward <> 0 THEN
		ptrExchgParamStationCommon^.T_DataValPercentAbs.rWorkingSpeedForward
			:=ABS(TOnlineChangeParameter.rWorkingSpeedForward/ptrProfileOnlineChange^.T_Max.rWorkingSpeedForward*100);
	ELSE ptrExchgParamStationCommon^.T_DataValPercentAbs.rWorkingSpeedForward:=-1; END_IF
	IF ptrProfileOnlineChange^.T_Max.rWorkingSpeedBackward <> 0 THEN
		ptrExchgParamStationCommon^.T_DataValPercentAbs.rWorkingSpeedBackward
			:=ABS(TOnlineChangeParameter.rWorkingSpeedBackward/ptrProfileOnlineChange^.T_Max.rWorkingSpeedBackward*100);
	ELSE ptrExchgParamStationCommon^.T_DataValPercentAbs.rWorkingSpeedBackward:=-1; END_IF
	IF ptrProfileOnlineChange^.T_Max.rForceDeflection <> 0 THEN
		rTmp:=TOnlineChangeParameter.rForceDeflection;
		rTmp:=rTmp/ptrProfileOnlineChange^.T_Max.rForceDeflection*100;
		ptrExchgParamStationCommon^.T_DataValPercentAbs.rForceDeflection:=ABS(rTmp);
	ELSE ptrExchgParamStationCommon^.T_DataValPercentAbs.rForceDeflection:=-1; END_IF
	IF ptrProfileOnlineChange^.T_Max.rTorqueLevelHC <> 0 THEN
		ptrExchgParamStationCommon^.T_DataValPercentAbs.rTorqueLevelHC
			:=ABS(TOnlineChangeParameter.rTorqueLevelHC/ptrProfileOnlineChange^.T_Max.rTorqueLevelHC*100);
	ELSE ptrExchgParamStationCommon^.T_DataValPercentAbs.rTorqueLevelHC:=-1; END_IF
	IF ptrProfileOnlineChange^.T_Min.rWorkingSpindleSpeed <> 0 THEN
		ptrExchgParamStationCommon^.T_DataValPercentAbs.rWorkingSpindleSpeed
			:=ABS(TOnlineChangeParameter.rWorkingSpindleSpeed/ptrProfileOnlineChange^.T_Min.rWorkingSpindleSpeed*100);
	ELSE ptrExchgParamStationCommon^.T_DataValPercentAbs.rWorkingSpindleSpeed:=-1; END_IF

(*  Update Rel perzent *)
	IF ptrProfileOnlineChangeLoad^.rWorkingOffsetBackward <> 0 THEN
		ptrExchgParamStationCommon^.T_DataValPercentRel.rWorkingOffsetBackward
			:=ABS(TOnlineChangeParameter.rWorkingOffsetBackward/ptrProfileOnlineChangeLoad^.rWorkingOffsetBackward*100);
	ELSE ptrExchgParamStationCommon^.T_DataValPercentRel.rWorkingOffsetBackward:=-1; END_IF
	IF ptrProfileOnlineChangeLoad^.rWorkingSpeedForward <> 0 THEN
		ptrExchgParamStationCommon^.T_DataValPercentRel.rWorkingSpeedForward
			:=ABS(TOnlineChangeParameter.rWorkingSpeedForward/ptrProfileOnlineChangeLoad^.rWorkingSpeedForward*100);
	ELSE ptrExchgParamStationCommon^.T_DataValPercentRel.rWorkingSpeedForward:=-1; END_IF
	IF ptrProfileOnlineChangeLoad^.rWorkingSpeedBackward <> 0 THEN
		ptrExchgParamStationCommon^.T_DataValPercentRel.rWorkingSpeedBackward
			:=ABS(TOnlineChangeParameter.rWorkingSpeedBackward/ptrProfileOnlineChangeLoad^.rWorkingSpeedBackward*100);
	ELSE ptrExchgParamStationCommon^.T_DataValPercentRel.rWorkingSpeedBackward:=-1; END_IF
	IF ptrProfileOnlineChangeLoad^.rForceDeflection <> 0 THEN
		rTmp:=TOnlineChangeParameter.rForceDeflection;
		rTmp:=rTmp/ptrProfileOnlineChangeLoad^.rForceDeflection*100;
		ptrExchgParamStationCommon^.T_DataValPercentRel.rForceDeflection:=ABS(rTmp);
	ELSE ptrExchgParamStationCommon^.T_DataValPercentRel.rForceDeflection:=-1; END_IF
	IF ptrProfileOnlineChangeLoad^.rTorqueLevelHC <> 0 THEN
		ptrExchgParamStationCommon^.T_DataValPercentRel.rTorqueLevelHC
			:=ABS(TOnlineChangeParameter.rTorqueLevelHC/ptrProfileOnlineChangeLoad^.rTorqueLevelHC*100);
	ELSE ptrExchgParamStationCommon^.T_DataValPercentRel.rTorqueLevelHC:=-1; END_IF
	IF ptrProfileOnlineChangeLoad^.rWorkingSpindleSpeed <> 0 THEN
		ptrExchgParamStationCommon^.T_DataValPercentRel.rWorkingSpindleSpeed
			:=ABS(TOnlineChangeParameter.rWorkingSpindleSpeed/ptrProfileOnlineChangeLoad^.rWorkingSpindleSpeed*100);
	ELSE ptrExchgParamStationCommon^.T_DataValPercentRel.rWorkingSpindleSpeed:=-1; END_IF

(* Min/Max value *)
	ptrExchgParamStationCommon^.T_Max:=ptrProfileOnlineChange^.T_Max;
	ptrExchgParamStationCommon^.T_Min:=ptrProfileOnlineChange^.T_Min;
END_FUNCTION

(* POU GENERAL/udiFct_FormatNumber, ST *)
FUNCTION udiFct_FormatNumber : UDINT
VAR_INPUT
	udiNumber:UDINT;
	iNumberLength:INT;
END_VAR
VAR
	sNumberToConvert: STRING(40);
	iCharCount: INT;
	sNumberConverted: STRING(40);
END_VAR
sNumberToConvert:=UDINT_TO_STRING(udiNumber);
iCharCount:=LEN(sNumberToConvert);
udiFct_FormatNumber:=0;
IF (iNumberLength > 0) THEN
	IF (iCharCount >= iNumberLength) THEN
		sNumberConverted:=MID(STR:=sNumberToConvert,LEN:=iNumberLength,POS:=iCharCount - iNumberLength + 1);
	ELSE
		sNumberConverted:=MID(STR:=sNumberToConvert,LEN:=iCharCount,POS:=1);
	END_IF;
	udiFct_FormatNumber:=STRING_TO_UDINT(sNumberConverted);
END_IF;
END_FUNCTION

(* POU PRG_LAYER5_VISU/FB_VISU/Function/bFct_SetAxisStat, ST *)
FUNCTION bFct_SetAxisStat : BYTE
(*Set/Reset bitxxx of StatusByte according to Bool-Input-State*)
VAR_INPUT
	xbit0			:BOOL;		(*Power*)
	xbit1			:BOOL;		(*Ref, 	Spez:@Spindle: busy*)
	xbit2			:BOOL;		(*Busyf, 	Spez:@Spindle: error*)
	xbit3			:BOOL;		(*Error*)
	xbit4			:BOOL;		(*HWlimNeg*)
	xbit5			:BOOL;		(*HWlimPos*)
	bState		:BYTE;		(*Use same Input byte as the output byte*)
END_VAR
VAR
END_VAR
bState.0:=xbit0 ;
bState.1:=xbit1 ;
bState.2:=xbit2 ;
bState.3:=xbit3 ;
bState.4:=xbit4 ;
bState.5:=xbit5 ;

bFct_SetAxisStat:= bState;
END_FUNCTION

(* POU PRG_LAYER5_VISU/FB_VISU/Function/bFct_SetCylStat, ST *)
FUNCTION bFct_SetCylStat : BYTE
(*Set/Reset bit0/ 1 of Byte according to Input-State*)
VAR_INPUT
	xON			:BOOL;
	xOFF		:BOOL;
	bState		:BYTE;
END_VAR
VAR
END_VAR
bState.0:=xOFF ;
bState.1:=xON ;

bFct_SetCylStat:= bState;
END_FUNCTION
